# EPICS substitutions: ISIS/lvexportApp/Db/userHost.substitutions
# Example substitutions file

file "db/dbExample1.db" {
    { user = "faa59Host" }
}

file db/dbExample2.db {
    pattern { user, no, scan }
        { "faa59Host", 1, "1 second" }
        { "faa59Host", 2, "2 second" }
        { "faa59Host", 3, "5 second" }
}
